PROGRAM MAIN
VAR
	testMethods		: FB_Methods;
	testGenerics	: FB_Generics<100>;
END_VAR

testMethods.MethodDefaultValue(1);

END_PROGRAM

(* stored: Version 1.1.0.1, ProductVersion 3.1.4026.6
   POU MAIN: Id {8712e83b-f585-4a61-82b9-804ce9b43d9b}, SpecialFunc None *)
